(* PLC project canopen_slave, beremiz beremiz 1 *)
(* stored: creationDateTime 2008-06-24T18:44:00, modificationDateTime 2020-06-03T22:09:12, language en-US *)

PROGRAM test_main
  VAR
    outvar AT %QW0.0.8192.0 : INT;
    invar AT %IW0.0.8193.0 : INT;
  END_VAR

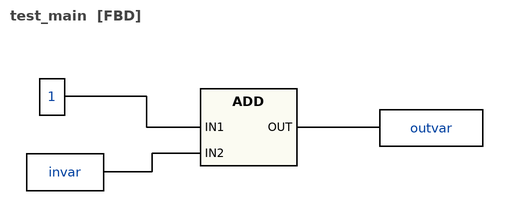
(* FBD diagram, written out as Structured Text *)
outvar := 1 + invar;
END_PROGRAM

CONFIGURATION conf
  RESOURCE res ON PLC
    TASK tache(INTERVAL := T#10ms, PRIORITY := 0);
    PROGRAM toto WITH tache : test_main;
  END_RESOURCE
END_CONFIGURATION
